(* Logix 5000 project; controller DCMGSG vendor 1 type 14 code 94 rev 20.12; software revision 20.01 *)
// Handles Scenario Generation I/O for DCMG.

TASK MainTask (continuous, watchdog 500 ms) : MainProgram

MODULES
   Local : vendor 1 type 14 code 94 (ICP 0, rev 20.12)
      SG_OB32_1 : 1756-OB32 (ICP 8, rev 3.3, Output RPI 20 ms)   // Digital output for DCMG Scenario Generator
      SG_OB32_2 : 1756-OB32 (ICP 9, rev 3.3, Output RPI 20 ms)   // Digital output for DCMG Scenario Generator. Signals 33 and up.
      EnvironmentSignals : 1756-OF4 (ICP 7, rev 1.1, Output RPI 12 ms)   // Signals for solar lamp dimming and turbine motor control.
      ETHERNET : 1756-EN2T (ICP 1, Ethernet 192.168.56.222, rev 3.1)
END_MODULES

VAR_GLOBAL   (* controller tags *)
   BRANCH_1_BUS_1_DISTAL_NC : BOOL;
   BRANCH_1_BUS_1_DISTAL_NC_ALIAS : ALIAS FOR Local:8:O.Data.22;
   BRANCH_1_BUS_1_DISTAL_NO : BOOL;
   BRANCH_1_BUS_1_DISTAL_NO_ALIAS : ALIAS FOR Local:8:O.Data.21;
   BRANCH_1_BUS_1_FAULT : BOOL;
   BRANCH_1_BUS_1_FAULT_ALIAS : ALIAS FOR Local:8:O.Data.23;
   BRANCH_1_BUS_1_LOAD_1_NC : BOOL;
   BRANCH_1_BUS_1_LOAD_1_NC_ALIAS : ALIAS FOR Local:8:O.Data.7;
   BRANCH_1_BUS_1_LOAD_1_NO : BOOL;
   BRANCH_1_BUS_1_LOAD_1_NO_ALIAS : ALIAS FOR Local:8:O.Data.6;
   BRANCH_1_BUS_1_LOAD_2_NC : BOOL;
   BRANCH_1_BUS_1_LOAD_2_NC_ALIAS : ALIAS FOR Local:8:O.Data.5;
   BRANCH_1_BUS_1_LOAD_2_NO : BOOL;
   BRANCH_1_BUS_1_LOAD_2_NO_ALIAS : ALIAS FOR Local:8:O.Data.4;
   BRANCH_1_BUS_1_LOAD_3_NC : BOOL;
   BRANCH_1_BUS_1_LOAD_3_NC_ALIAS : ALIAS FOR Local:8:O.Data.0;
   BRANCH_1_BUS_1_LOAD_3_NO : BOOL;
   BRANCH_1_BUS_1_LOAD_3_NO_ALIAS : ALIAS FOR Local:8:O.Data.3;
   BRANCH_1_BUS_1_PROXIMAL_NC : BOOL;
   BRANCH_1_BUS_1_PROXIMAL_NC_ALIAS : ALIAS FOR Local:8:O.Data.2;
   BRANCH_1_BUS_1_PROXIMAL_NO : BOOL;
   BRANCH_1_BUS_1_PROXIMAL_NO_ALIAS : ALIAS FOR Local:8:O.Data.1;
   BRANCH_1_BUS_2_DISTAL_NC : BOOL;
   BRANCH_1_BUS_2_DISTAL_NC_ALIAS : ALIAS FOR Local:9:O.Data.4;
   BRANCH_1_BUS_2_DISTAL_NO : BOOL;
   BRANCH_1_BUS_2_DISTAL_NO_ALIAS : ALIAS FOR Local:9:O.Data.5;
   BRANCH_1_BUS_2_FAULT : BOOL;
   BRANCH_1_BUS_2_FAULT_ALIAS : ALIAS FOR Local:9:O.Data.8;
   BRANCH_1_BUS_2_LOAD_1_NC : BOOL;
   BRANCH_1_BUS_2_LOAD_1_NC_ALIAS : ALIAS FOR Local:8:O.Data.31;
   BRANCH_1_BUS_2_LOAD_1_NO : BOOL;
   BRANCH_1_BUS_2_LOAD_1_NO_ALIAS : ALIAS FOR Local:9:O.Data.0;
   BRANCH_1_BUS_2_LOAD_2_NC : BOOL;
   BRANCH_1_BUS_2_LOAD_2_NC_ALIAS : ALIAS FOR Local:9:O.Data.1;
   BRANCH_1_BUS_2_LOAD_2_NO : BOOL;
   BRANCH_1_BUS_2_LOAD_2_NO_ALIAS : ALIAS FOR Local:9:O.Data.2;
   BRANCH_1_BUS_2_LOAD_3_NC : BOOL;
   BRANCH_1_BUS_2_LOAD_3_NC_ALIAS : ALIAS FOR Local:9:O.Data.6;
   BRANCH_1_BUS_2_LOAD_3_NO : BOOL;
   BRANCH_1_BUS_2_LOAD_3_NO_ALIAS : ALIAS FOR Local:9:O.Data.7;
   BRANCH_1_BUS_2_PROXIMAL_NC : BOOL;
   BRANCH_1_BUS_2_PROXIMAL_NC_ALIAS : ALIAS FOR Local:8:O.Data.25;
   BRANCH_1_BUS_2_PROXIMAL_NO : BOOL;
   BRANCH_1_BUS_2_PROXIMAL_NO_ALIAS : ALIAS FOR Local:8:O.Data.26;
   BRANCH_1_INTERCONNECT_1_FAULT : BOOL;
   BRANCH_1_INTERCONNECT_1_FAULT_ALIAS : ALIAS FOR Local:8:O.Data.24;
   BRANCH_1_INTERCONNECT_2_FAULT : BOOL;
   BRANCH_1_INTERCONNECT_2_FAULT_ALIAS : ALIAS FOR Local:9:O.Data.9;
   BRANCH_2_BUS_1_DISTAL_NC : BOOL;
   BRANCH_2_BUS_1_DISTAL_NC_ALIAS : ALIAS FOR Local:8:O.Data.9;
   BRANCH_2_BUS_1_DISTAL_NO : BOOL;
   BRANCH_2_BUS_1_DISTAL_NO_ALIAS : ALIAS FOR Local:8:O.Data.10;
   BRANCH_2_BUS_1_FAULT : BOOL;
   BRANCH_2_BUS_1_FAULT_ALIAS : ALIAS FOR Local:8:O.Data.29;
   BRANCH_2_BUS_1_LOAD_1_NC : BOOL;
   BRANCH_2_BUS_1_LOAD_1_NC_ALIAS : ALIAS FOR Local:8:O.Data.15;
   BRANCH_2_BUS_1_LOAD_1_NO : BOOL;
   BRANCH_2_BUS_1_LOAD_1_NO_ALIAS : ALIAS FOR Local:8:O.Data.8;
   BRANCH_2_BUS_1_LOAD_2_NC : BOOL;
   BRANCH_2_BUS_1_LOAD_2_NC_ALIAS : ALIAS FOR Local:8:O.Data.16;
   BRANCH_2_BUS_1_LOAD_2_NO : BOOL;
   BRANCH_2_BUS_1_LOAD_2_NO_ALIAS : ALIAS FOR Local:8:O.Data.14;
   BRANCH_2_BUS_1_LOAD_3_NC : BOOL;
   BRANCH_2_BUS_1_LOAD_3_NC_ALIAS : ALIAS FOR Local:8:O.Data.18;
   BRANCH_2_BUS_1_LOAD_3_NO : BOOL;
   BRANCH_2_BUS_1_LOAD_3_NO_ALIAS : ALIAS FOR Local:8:O.Data.17;
   BRANCH_2_BUS_1_PROXIMAL_NC : BOOL;
   BRANCH_2_BUS_1_PROXIMAL_NC_ALIAS : ALIAS FOR Local:8:O.Data.11;
   BRANCH_2_BUS_1_PROXIMAL_NO : BOOL;
   BRANCH_2_BUS_1_PROXIMAL_NO_ALIAS : ALIAS FOR Local:8:O.Data.12;
   BRANCH_2_BUS_2_DISTAL_NC : BOOL;
   BRANCH_2_BUS_2_DISTAL_NC_ALIAS : ALIAS FOR Local:9:O.Data.13;
   BRANCH_2_BUS_2_DISTAL_NO : BOOL;
   BRANCH_2_BUS_2_DISTAL_NO_ALIAS : ALIAS FOR Local:9:O.Data.14;
   BRANCH_2_BUS_2_FAULT : BOOL;
   BRANCH_2_BUS_2_FAULT_ALIAS : ALIAS FOR Local:9:O.Data.11;
   BRANCH_2_BUS_2_LOAD_1_NC : BOOL;
   BRANCH_2_BUS_2_LOAD_1_NC_ALIAS : ALIAS FOR Local:9:O.Data.20;
   BRANCH_2_BUS_2_LOAD_1_NO : BOOL;
   BRANCH_2_BUS_2_LOAD_1_NO_ALIAS : ALIAS FOR Local:9:O.Data.12;
   BRANCH_2_BUS_2_LOAD_2_NC : BOOL;
   BRANCH_2_BUS_2_LOAD_2_NC_ALIAS : ALIAS FOR Local:9:O.Data.18;
   BRANCH_2_BUS_2_LOAD_2_NO : BOOL;
   BRANCH_2_BUS_2_LOAD_2_NO_ALIAS : ALIAS FOR Local:9:O.Data.19;
   BRANCH_2_BUS_2_LOAD_3_NC : BOOL;
   BRANCH_2_BUS_2_LOAD_3_NC_ALIAS : ALIAS FOR Local:9:O.Data.16;
   BRANCH_2_BUS_2_LOAD_3_NO : BOOL;
   BRANCH_2_BUS_2_LOAD_3_NO_ALIAS : ALIAS FOR Local:9:O.Data.17;
   BRANCH_2_BUS_2_PROXIMAL_NC : BOOL;
   BRANCH_2_BUS_2_PROXIMAL_NC_ALIAS : ALIAS FOR Local:8:O.Data.28;
   BRANCH_2_BUS_2_PROXIMAL_NO : BOOL;
   BRANCH_2_BUS_2_PROXIMAL_NO_ALIAS : ALIAS FOR Local:8:O.Data.27;
   BRANCH_2_INTERCONNECT_1_FAULT : BOOL;
   BRANCH_2_INTERCONNECT_1_FAULT_ALIAS : ALIAS FOR Local:8:O.Data.30;
   BRANCH_2_INTERCONNECT_2_FAULT : BOOL;
   BRANCH_2_INTERCONNECT_2_FAULT_ALIAS : ALIAS FOR Local:9:O.Data.10;
   CROSSTIE_1_NC : BOOL;
   CROSSTIE_1_NC_ALIAS : ALIAS FOR Local:8:O.Data.20;
   CROSSTIE_1_NO : BOOL;
   CROSSTIE_1_NO_ALIAS : ALIAS FOR Local:8:O.Data.19;
   CROSSTIE_2_NC : BOOL;
   CROSSTIE_2_NC_ALIAS : ALIAS FOR Local:9:O.Data.3;
   CROSSTIE_2_NO : BOOL;
   CROSSTIE_2_NO_ALIAS : ALIAS FOR Local:9:O.Data.15;
   MAIN_BUS_FAULT : BOOL;
   MAIN_BUS_FAULT_ALIAS : ALIAS FOR Local:8:O.Data.13;
   SolarSetpoint1Alias : REAL;
   SolarSetpoint1Alias_ALIAS : ALIAS FOR Local:7:O.Ch0Data;
   SolarSetpoint2Alias : REAL;
   SolarSetpoint2Alias_ALIAS : ALIAS FOR Local:7:O.Ch1Data;
   SOURCE_1_NC : BOOL;
   SOURCE_1_NC_ALIAS : ALIAS FOR Local:9:O.Data.21;
   SOURCE_2_NC : BOOL;
   SOURCE_2_NC_ALIAS : ALIAS FOR Local:9:O.Data.22;
   SOURCE_3_NC : BOOL;
   SOURCE_3_NC_ALIAS : ALIAS FOR Local:9:O.Data.23;
   SOURCE_4_NC : BOOL;
   SOURCE_4_NC_ALIAS : ALIAS FOR Local:9:O.Data.24;
   SOURCE_5_NC : BOOL;
   SOURCE_5_NC_ALIAS : ALIAS FOR Local:9:O.Data.25;
   SOURCE_6_NC : BOOL;
   SOURCE_6_NC_ALIAS : ALIAS FOR Local:9:O.Data.26;
END_VAR

PROGRAM MainProgram   (* main routine MainRoutine *)

ROUTINE MainRoutine   (* ladder *)
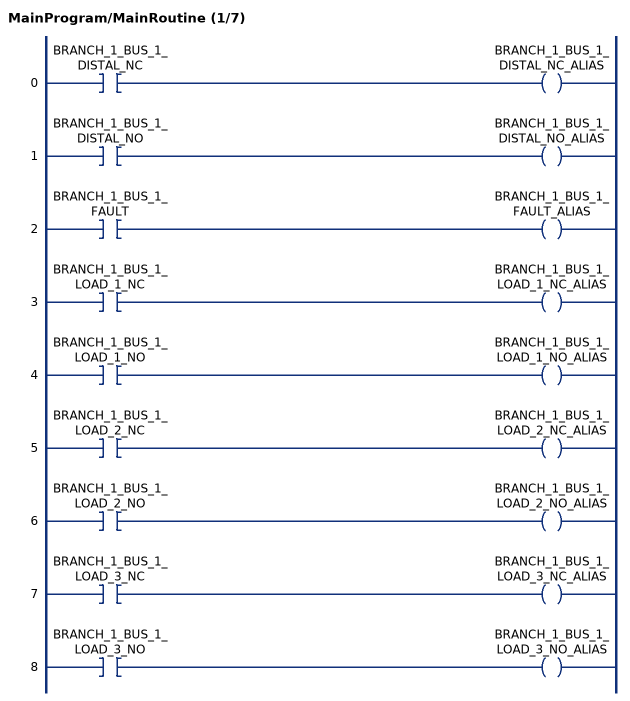
   0: XIC(BRANCH_1_BUS_1_DISTAL_NC)OTE(BRANCH_1_BUS_1_DISTAL_NC_ALIAS);
   1: XIC(BRANCH_1_BUS_1_DISTAL_NO)OTE(BRANCH_1_BUS_1_DISTAL_NO_ALIAS);
   2: XIC(BRANCH_1_BUS_1_FAULT)OTE(BRANCH_1_BUS_1_FAULT_ALIAS);
   3: XIC(BRANCH_1_BUS_1_LOAD_1_NC)OTE(BRANCH_1_BUS_1_LOAD_1_NC_ALIAS);
   4: XIC(BRANCH_1_BUS_1_LOAD_1_NO)OTE(BRANCH_1_BUS_1_LOAD_1_NO_ALIAS);
   5: XIC(BRANCH_1_BUS_1_LOAD_2_NC)OTE(BRANCH_1_BUS_1_LOAD_2_NC_ALIAS);
   6: XIC(BRANCH_1_BUS_1_LOAD_2_NO)OTE(BRANCH_1_BUS_1_LOAD_2_NO_ALIAS);
   7: XIC(BRANCH_1_BUS_1_LOAD_3_NC)OTE(BRANCH_1_BUS_1_LOAD_3_NC_ALIAS);
   8: XIC(BRANCH_1_BUS_1_LOAD_3_NO)OTE(BRANCH_1_BUS_1_LOAD_3_NO_ALIAS);
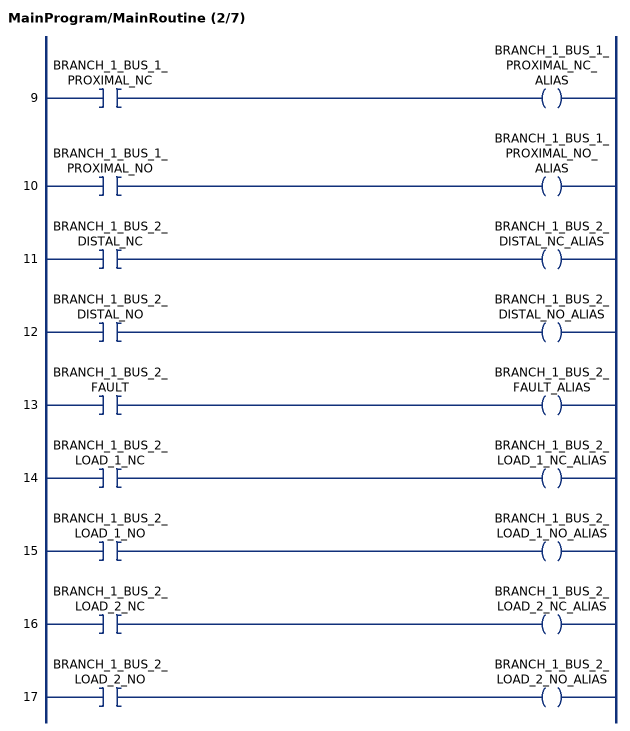
   9: XIC(BRANCH_1_BUS_1_PROXIMAL_NC)OTE(BRANCH_1_BUS_1_PROXIMAL_NC_ALIAS);
   10: XIC(BRANCH_1_BUS_1_PROXIMAL_NO)OTE(BRANCH_1_BUS_1_PROXIMAL_NO_ALIAS);
   11: XIC(BRANCH_1_BUS_2_DISTAL_NC)OTE(BRANCH_1_BUS_2_DISTAL_NC_ALIAS);
   12: XIC(BRANCH_1_BUS_2_DISTAL_NO)OTE(BRANCH_1_BUS_2_DISTAL_NO_ALIAS);
   13: XIC(BRANCH_1_BUS_2_FAULT)OTE(BRANCH_1_BUS_2_FAULT_ALIAS);
   14: XIC(BRANCH_1_BUS_2_LOAD_1_NC)OTE(BRANCH_1_BUS_2_LOAD_1_NC_ALIAS);
   15: XIC(BRANCH_1_BUS_2_LOAD_1_NO)OTE(BRANCH_1_BUS_2_LOAD_1_NO_ALIAS);
   16: XIC(BRANCH_1_BUS_2_LOAD_2_NC)OTE(BRANCH_1_BUS_2_LOAD_2_NC_ALIAS);
   17: XIC(BRANCH_1_BUS_2_LOAD_2_NO)OTE(BRANCH_1_BUS_2_LOAD_2_NO_ALIAS);
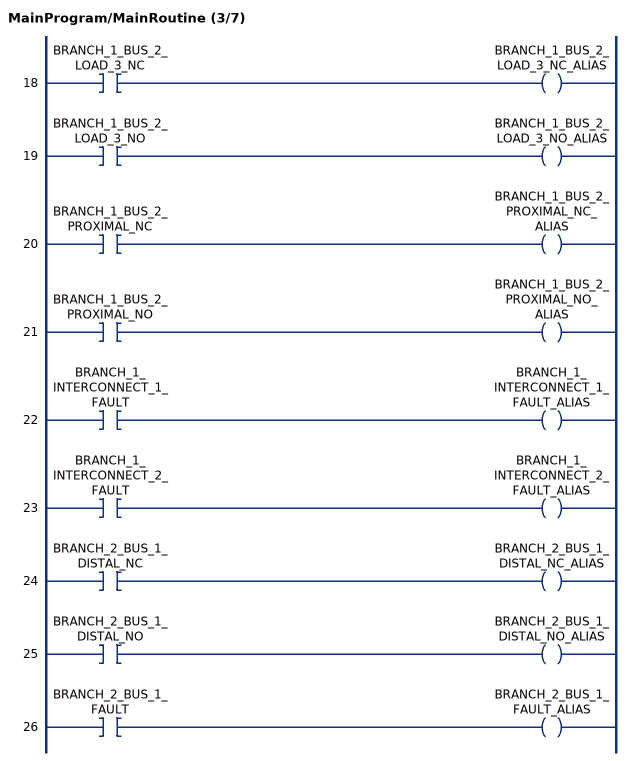
   18: XIC(BRANCH_1_BUS_2_LOAD_3_NC)OTE(BRANCH_1_BUS_2_LOAD_3_NC_ALIAS);
   19: XIC(BRANCH_1_BUS_2_LOAD_3_NO)OTE(BRANCH_1_BUS_2_LOAD_3_NO_ALIAS);
   20: XIC(BRANCH_1_BUS_2_PROXIMAL_NC)OTE(BRANCH_1_BUS_2_PROXIMAL_NC_ALIAS);
   21: XIC(BRANCH_1_BUS_2_PROXIMAL_NO)OTE(BRANCH_1_BUS_2_PROXIMAL_NO_ALIAS);
   22: XIC(BRANCH_1_INTERCONNECT_1_FAULT)OTE(BRANCH_1_INTERCONNECT_1_FAULT_ALIAS);
   23: XIC(BRANCH_1_INTERCONNECT_2_FAULT)OTE(BRANCH_1_INTERCONNECT_2_FAULT_ALIAS);
   24: XIC(BRANCH_2_BUS_1_DISTAL_NC)OTE(BRANCH_2_BUS_1_DISTAL_NC_ALIAS);
   25: XIC(BRANCH_2_BUS_1_DISTAL_NO)OTE(BRANCH_2_BUS_1_DISTAL_NO_ALIAS);
   26: XIC(BRANCH_2_BUS_1_FAULT)OTE(BRANCH_2_BUS_1_FAULT_ALIAS);
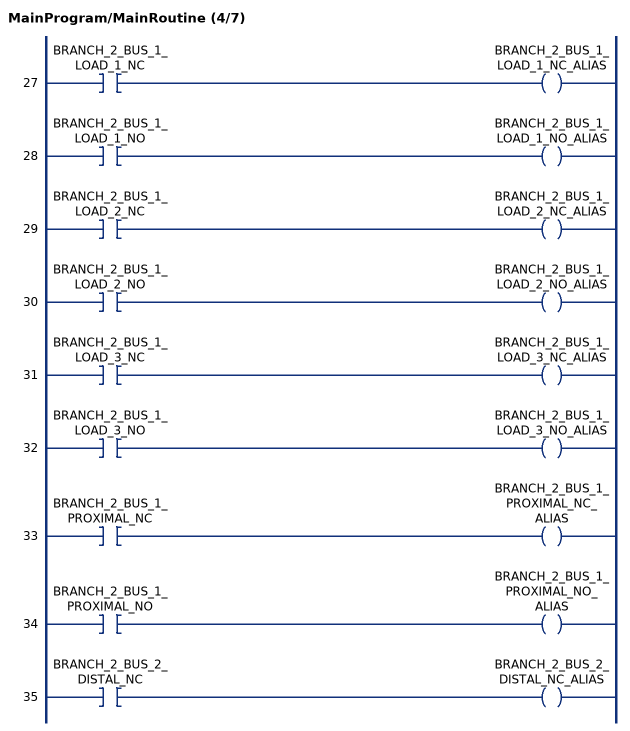
   27: XIC(BRANCH_2_BUS_1_LOAD_1_NC)OTE(BRANCH_2_BUS_1_LOAD_1_NC_ALIAS);
   28: XIC(BRANCH_2_BUS_1_LOAD_1_NO)OTE(BRANCH_2_BUS_1_LOAD_1_NO_ALIAS);
   29: XIC(BRANCH_2_BUS_1_LOAD_2_NC)OTE(BRANCH_2_BUS_1_LOAD_2_NC_ALIAS);
   30: XIC(BRANCH_2_BUS_1_LOAD_2_NO)OTE(BRANCH_2_BUS_1_LOAD_2_NO_ALIAS);
   31: XIC(BRANCH_2_BUS_1_LOAD_3_NC)OTE(BRANCH_2_BUS_1_LOAD_3_NC_ALIAS);
   32: XIC(BRANCH_2_BUS_1_LOAD_3_NO)OTE(BRANCH_2_BUS_1_LOAD_3_NO_ALIAS);
   33: XIC(BRANCH_2_BUS_1_PROXIMAL_NC)OTE(BRANCH_2_BUS_1_PROXIMAL_NC_ALIAS);
   34: XIC(BRANCH_2_BUS_1_PROXIMAL_NO)OTE(BRANCH_2_BUS_1_PROXIMAL_NO_ALIAS);
   35: XIC(BRANCH_2_BUS_2_DISTAL_NC)OTE(BRANCH_2_BUS_2_DISTAL_NC_ALIAS);
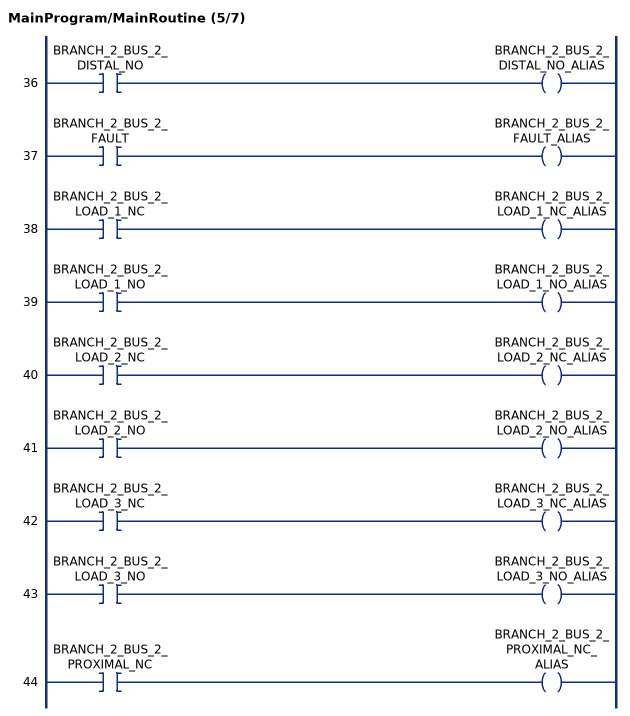
   36: XIC(BRANCH_2_BUS_2_DISTAL_NO)OTE(BRANCH_2_BUS_2_DISTAL_NO_ALIAS);
   37: XIC(BRANCH_2_BUS_2_FAULT)OTE(BRANCH_2_BUS_2_FAULT_ALIAS);
   38: XIC(BRANCH_2_BUS_2_LOAD_1_NC)OTE(BRANCH_2_BUS_2_LOAD_1_NC_ALIAS);
   39: XIC(BRANCH_2_BUS_2_LOAD_1_NO)OTE(BRANCH_2_BUS_2_LOAD_1_NO_ALIAS);
   40: XIC(BRANCH_2_BUS_2_LOAD_2_NC)OTE(BRANCH_2_BUS_2_LOAD_2_NC_ALIAS);
   41: XIC(BRANCH_2_BUS_2_LOAD_2_NO)OTE(BRANCH_2_BUS_2_LOAD_2_NO_ALIAS);
   42: XIC(BRANCH_2_BUS_2_LOAD_3_NC)OTE(BRANCH_2_BUS_2_LOAD_3_NC_ALIAS);
   43: XIC(BRANCH_2_BUS_2_LOAD_3_NO)OTE(BRANCH_2_BUS_2_LOAD_3_NO_ALIAS);
   44: XIC(BRANCH_2_BUS_2_PROXIMAL_NC)OTE(BRANCH_2_BUS_2_PROXIMAL_NC_ALIAS);
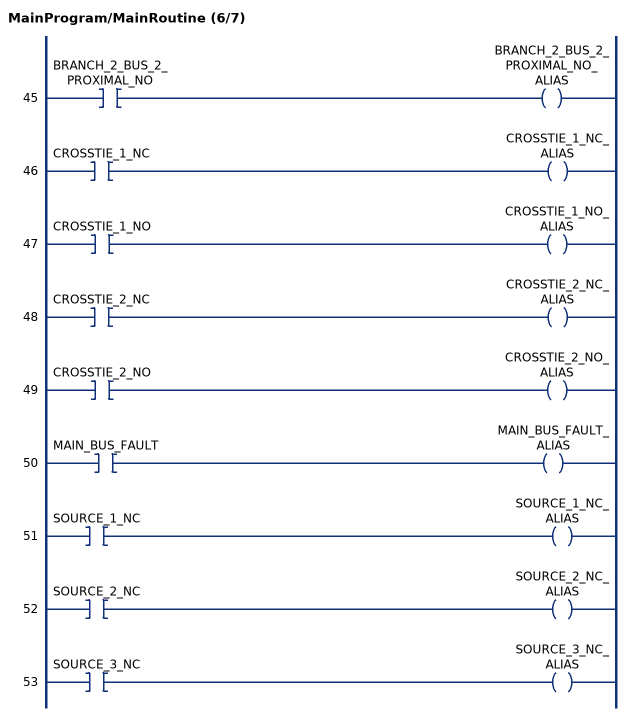
   45: XIC(BRANCH_2_BUS_2_PROXIMAL_NO)OTE(BRANCH_2_BUS_2_PROXIMAL_NO_ALIAS);
   46: XIC(CROSSTIE_1_NC)OTE(CROSSTIE_1_NC_ALIAS);
   47: XIC(CROSSTIE_1_NO)OTE(CROSSTIE_1_NO_ALIAS);
   48: XIC(CROSSTIE_2_NC)OTE(CROSSTIE_2_NC_ALIAS);
   49: XIC(CROSSTIE_2_NO)OTE(CROSSTIE_2_NO_ALIAS);
   50: XIC(MAIN_BUS_FAULT)OTE(MAIN_BUS_FAULT_ALIAS);
   51: XIC(SOURCE_1_NC)OTE(SOURCE_1_NC_ALIAS);
   52: XIC(SOURCE_2_NC)OTE(SOURCE_2_NC_ALIAS);
   53: XIC(SOURCE_3_NC)OTE(SOURCE_3_NC_ALIAS);
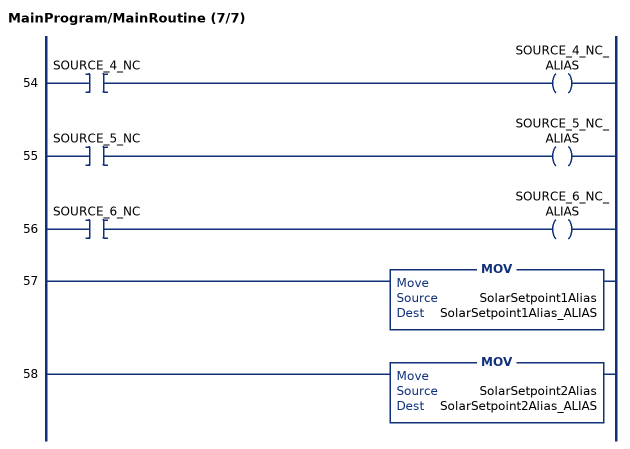
   54: XIC(SOURCE_4_NC)OTE(SOURCE_4_NC_ALIAS);
   55: XIC(SOURCE_5_NC)OTE(SOURCE_5_NC_ALIAS);
   56: XIC(SOURCE_6_NC)OTE(SOURCE_6_NC_ALIAS);
   57: MOV(SolarSetpoint1Alias,SolarSetpoint1Alias_ALIAS);
   58: MOV(SolarSetpoint2Alias,SolarSetpoint2Alias_ALIAS);
END_ROUTINE
END_PROGRAM
